// TwinCAT 3 PLC project PLC
// Title: NC Sample Code using Tria-Link
// Company: Triamec Motion AG
// Author: Triamec Motion AG
// Description: NC Sample Code using Tria-Link
// ProgramVersion: 3.1.4024.0
// libraries:
//   Tc2_MC2, * (Beckhoff Automation GmbH)
//   Tc2_Standard, * (Beckhoff Automation GmbH)
//   Tc2_System, * (Beckhoff Automation GmbH)
//   Tc3_Module, * (Beckhoff Automation GmbH)
//   Triamec, * (Triamec Motion AG)
// project tree:
//   / Fast_Task.TcTTO, Slow_Task.TcTTO
//   POUs/ NC_Axis.TcPOU, Triamec_GVL.TcGVL, MAIN.TcPOU, MAIN_FAST.TcPOU
// real-time tasks:
//   TASK Slow_Task: cycle T#2500us, priority 6, ADS port 350
// motion (NC):
//   TASK NC-Task 1 SAF: cycle T#500us, priority 4, ADS port 501
//   TASK NC-Task 1 SVB: cycle T#10ms, priority 10, ADS port 511
//   AXIS Axis X (id 1)
//     OtherSettings: AllowMotionCmdToSlave=true
//     encoder EncType=8
//       EncPara: ScaleFactorNumerator=1e-06, MaxCount=#xffffffff
//         Inc: RefSoftSyncMask=#xffffffff
//     drive DrvType=9
//       DrvPara: MaxCount=#xffffffff
//         Analog: VeloScale=6, TorqueSetpointScale=10, ScaleFactorActTorque=0.1
//         TimeComp: TaskDelayCycles=1
//     controller CtrType=9
//       CtrPara: PriorControlFactor=1
//         Observer: BandWidth=20
//   AXIS Axis Y (id 2)
//     OtherSettings: AllowMotionCmdToSlave=true
//     encoder EncType=8
//       EncPara: ScaleFactorNumerator=1e-06, MaxCount=#xffffffff
//         Inc: RefSoftSyncMask=#xffffffff
//     drive DrvType=9
//       DrvPara: MaxCount=#xffffffff
//         Analog: VeloScale=6, TorqueSetpointScale=10, ScaleFactorActTorque=0.1
//         TimeComp: TaskDelayCycles=1
//     controller CtrType=9
//       CtrPara: PriorControlFactor=1
//         Observer: BandWidth=20
// I/O:
//   DEVICE TriaLink (NOV-DP-RAM)
// variable links:
//   PLC/PLC Instance <-> NC-Task 1 SAF/Axes/Axis X
//     Fast_Task Inputs/MAIN.Axes[1].PosCmd <-> Drive/Outputs/Out/nDataOut1
//     Fast_Task Outputs/MAIN.Axes[1].PosAct <-> Enc/Inputs/In/nDataIn1
//     Slow_Task Inputs/MAIN.Axes[1].nciAxis.NcToPlc <-> Outputs/ToPlc
//     Slow_Task Outputs/MAIN.Axes[1].State1 <-> Drive/Inputs/In/nState1
//     Slow_Task Outputs/MAIN.Axes[1].State4 <-> Drive/Inputs/In/nState4
//     Slow_Task Outputs/MAIN.Axes[1].nciAxis.PlcToNc <-> Inputs/FromPlc
//   PLC/PLC Instance <-> NC-Task 1 SAF/Axes/Axis Y
//     Fast_Task Inputs/MAIN.Axes[2].PosCmd <-> Drive/Outputs/Out/nDataOut1
//     Fast_Task Outputs/MAIN.Axes[2].PosAct <-> Enc/Inputs/In/nDataIn1
//     Slow_Task Inputs/MAIN.Axes[2].nciAxis.NcToPlc <-> Outputs/ToPlc
//     Slow_Task Outputs/MAIN.Axes[2].State1 <-> Drive/Inputs/In/nState1
//     Slow_Task Outputs/MAIN.Axes[2].State4 <-> Drive/Inputs/In/nState4
//     Slow_Task Outputs/MAIN.Axes[2].nciAxis.PlcToNc <-> Inputs/FromPlc

CONFIGURATION PLC
    RESOURCE PLC ON TwinCAT3
        TASK Fast_Task(INTERVAL := T#500us, PRIORITY := 4);
        TASK Slow_Task(INTERVAL := T#2500us, PRIORITY := 6);
        PROGRAM MAIN_FAST WITH Fast_Task : MAIN_FAST;
        PROGRAM MAIN WITH Slow_Task : MAIN;
    END_RESOURCE
END_CONFIGURATION

// ---- POUs/Triamec_GVL.TcGVL
VAR_GLOBAL
	gEnableTrialink : BOOL; 	(* variable to enable Tria-Link *)
	gEnableAxes : BOOL; 		(* variable to enable all axes *)
	gResetAxes : BOOL; 			(* variable to reset all axes *)
	gCommunicationReady : BOOL; (* indicator for Tria-Link and axes readiness *)
END_VAR

// ---- POUs/MAIN_FAST.TcPOU
PROGRAM MAIN_FAST
VAR
	i : USINT; (* counter variable *)
END_VAR

(* --------------------------------------------- *)
(* Triamec Motion AG, 6340 Baar, Switzerland     *)
(* Sample Code may be adapted to customer need   *)
(* --------------------------------------------- *)

(* Tria-Link cyclic fast call *)
MAIN.Trialink.CallFast();

(* CNC axis cyclic fast call *)
FOR i := 1 TO MAIN.cAxes DO
	MAIN.Axes[i].Fast();
END_FOR

END_PROGRAM

// ---- POUs/MAIN.TcPOU
PROGRAM MAIN
VAR CONSTANT
	cAxes			: USINT := 2; (* Number of axes in use *)
END_VAR

VAR
	Trialink : Triamec.TL_Trialink2; 		(* the Tria-Link adapter *)
	Axes : ARRAY [1..cAxes] OF NC_Axis; 	(* the extended triamec axis object with link to the NC *)
	
	initDone : BOOL;	(* initialization done *)
	i : USINT; 			(* counter variable *)
END_VAR

(* ------------------------------------------- *)
(* Triamec Motion AG, 6340 Baar, Switzerland   *)
(* Sample Code may be adapted to customer need *)
(* ------------------------------------------- *)

(* Tria-Link and Axes configuration *)
IF NOT initDone THEN
	initDone := Config();
END_IF

(* Tria-Link cyclic call*)
Trialink.Execute := gEnableTrialink;
Trialink.CallSlow();
gCommunicationReady := gEnableTrialink AND NOT Trialink.Error;

(* Axes cyclic call *)
FOR i := 1 TO cAxes DO
	Axes[i].iAxis := i;				// logical axis number
	Axes[i].reset := gResetAxes; 	// reset drive errors
	Axes[i].enable := gEnableAxes; 	// set enable / disable
	Axes[i].couple := TRUE;			// couple drive to CNC pathplanner
	Axes[i](Trialink := Trialink); 	// cyclic call of cnc axes
	gCommunicationReady	:= gCommunicationReady AND Axes[i].ready;
END_FOR

METHOD Config : BOOL
(* Tria-Link configuration *)
Trialink.Config.nDevId := 1; // NOV-DP-RAM Id, see TwinCAT System Manager (I/0 > Devices > TriaLink) 
Trialink.Config.TcEventEnable := TRUE;

(* Axes configuration *)
(* ---------- Axis 1 ---------- *)
Axes[1].inc_per_unit 		:= 1000000; // scale between CNC and PLC
Axes[1].Config.Simulate   	:= FALSE;
Axes[1].Config.Station    	:= 10;		// The drive address
Axes[1].Config.SubAxis    	:= TL_Config.SubAxis.FirstAxis; // first or second axis of a two axes drive
Axes[1].Config.GearFactor 	:= 1;		// multiplication factor of position and velocity data
Axes[1].Config.ModuloWrap 	:= 0;		// modulo wrap for rotation axes
Axes[1].referencePos 		:= 0.0;		// reference position to which the axis is set after homing
	
(* ---------- Axis 2 ---------- *)
Axes[2].inc_per_unit 		:= 1000000; // scale between CNC and PLC
Axes[2].Config.Simulate   	:= TRUE;
Axes[2].Config.Station    	:= 10;		// The drive address
Axes[2].Config.SubAxis    	:= TL_Config.SubAxis.SecondAxis; // first or second axis of a two axes drive
Axes[2].Config.GearFactor 	:= 1;		// multiplication factor of position and velocity data
Axes[2].Config.ModuloWrap 	:= 0;		// modulo wrap for rotation axes
Axes[2].referencePos 		:= 0.0; 	// reference position to which the axis is set after homing

Config := TRUE;
END_METHOD

END_PROGRAM

// ---- POUs/NC_Axis.TcPOU
FUNCTION_BLOCK NC_Axis EXTENDS Triamec.TL_Axis2
VAR_IN_OUT
	Trialink	: Triamec.TL_Trialink2; (* the Tria-Link adapter *)
END_VAR
VAR_INPUT
	nciAxis	: AXIS_REF; 			(* axis reference *)
	inc_per_unit : LREAL := 1E7; 	(* use 10000 inc/deg or 1E7 inc/m *)
END_VAR
VAR
		 
	State1	AT %Q*		: BYTE; 	(* NC > Axis > Drive > Inputs > nState1 *)
	State4	AT %Q*		: BYTE; 	(* NC > Axis > Drive > Inputs > nState4 *)
	PosCmd	AT %I*		: DWORD;	(* NC > Axis > Drive > Outputs > nDataOut1 *)
	PosAct	AT %Q*		: DWORD;	(* NC > Axis > Enc > Inputs > nDataIn1 *)
	
	FB_MC_Power			: MC_Power;
	FB_MC_Reset			: MC_Reset;
	FB_Reset1			: R_TRIG;
	FB_Reset2			: R_TRIG;
	
	MessageHandler	: TL_AxisMessageHandler;	// provides corresponding message string
	TcEventLib		: TL_TwinCatError;
	TcEventDrv		: TL_TwinCatError;
END_VAR

(* --------------------------------------------- *)
(* Triamec Motion AG, 6340 Baar, Switzerland     *)
(* Sample Code may be adapted to customer need   *)
(* --------------------------------------------- *)

SUPER^.CallSlow(Trialink := THIS^.Trialink);

(*
  Sercos Status Word
  Status1 = 16#4? DriveOn  
  Status1 = 16#8? Feedhold  
  Status1 = 16#C? TorquePermission  
*)
IF NOT enable THEN
	State1 :=    0;
	State4 :=    4;
ELSIF coupled THEN
	State1 :=16#C8;
	State4 :=    4;
ELSE
	State1 :=16#C0;
	State4 :=    4;
END_IF
IF referenced THEN
	State1 :=    State1 + 1;
END_IF

(* enable the NCI module *)
FB_MC_Power.Enable			:= enable;
FB_MC_Power.Enable_Negative	:= TRUE;
FB_MC_Power.Enable_Positive	:= TRUE;
FB_MC_Power.Override		:= 100;
FB_MC_Power(Axis := nciAxis);

FB_Reset1(CLK:=NOT followMe);
FB_Reset2(CLK:=Reset);
FB_MC_Reset.Execute			:= FB_Reset1.Q OR FB_Reset2.Q;
FB_MC_Reset(Axis := nciAxis);

(* This reads the drive message string into messageHandler.messageString and then sets messageHandler.done *)
MessageHandler.execute := messageId >= TL_Message.Error; // show only errors
MessageHandler(axis:=MC_axis, Trialink:=Trialink);

(* This generates a TwinCAT event in case of an axis library error and an axis drive error *)
TcEventLib.Execute	:= Trialink.Done AND NOT (Trialink.Error OR MC_axis.simulate);
TcEventLib.errorId	:= MC_axis.errorId;
TcEventLib.source	:= TL_EventSourceId.AxisLib; // See source entry in file triamecEventsTrialink.xml
TcEventLib.par1	:= MC_axis.iAxis;
TcEventLib();

TcEventDrv.Execute	:= TcEventLib.Execute AND MC_axis.messageId>=TL_Message.Error; // show only errors 
TcEventDrv.errorId	:= MC_axis.messageId;
TcEventDrv.source	:= TL_EventSourceId.AxisDrive; // See source entry in the file triamecEventsDrive.xml
TcEventDrv.par1	:= MC_axis.iAxis;
TcEventDrv();

METHOD Fast
VAR
	positionAct : LREAL; (* actual position *)
END_VAR
// The warning can be disabled here as the user is aware of the risk that the reference may not be valid by checking its validity
{warning disable C0371}

// Checking the VAR_IN_OUT reference, leave the current method in case of invalid reference
IF NOT __ISVALIDREF(Trialink) THEN
     RETURN;
END_IF

(* get the coordinates from the NC/CNC and write it to the drive *)
fastPositionCmd := DINT_TO_LREAL(DWORD_TO_DINT(PosCmd)) / inc_per_unit;
SUPER^.CallFast( Trialink := Trialink );

(* get the actual position from the drive and pass it to NC *)
positionAct := ActualPositionFast(Trialink := Trialink);
(* coerse position to DINT range *)
IF ABS(positionAct * inc_per_unit) < 16#7FFFFFFF  THEN
	PosAct := DINT_TO_DWORD(LREAL_TO_DINT(positionAct * inc_per_unit));
ELSIF positionAct < 0 THEN
	PosAct := 16#80000000;
ELSE
	PosAct := 16#7FFFFFFF;
END_IF

// The warning may be restored at the end of the access area
{warning restore C0371}
END_METHOD

END_FUNCTION_BLOCK
